TYPE EL3xx8 :
STRUCT
	ch1		:INT;
	ch2		:INT;
	ch3		:INT;
	ch4		:INT;
	ch5		:INT;
	ch6		:INT;
	ch7		:INT;
	ch8		:INT;
END_STRUCT
END_TYPE

(* stored: Version 1.1.0.1, ProductVersion 3.1.4024.12
   DUT EL3xx8: Id {b0e7ae9c-3e87-4821-9170-0ce7ba62b0c7} *)
